% RSLogix 500 project XLT_EXP_BOTTOM.RSS, saved by version 11.00.00.00 %
PROJECT "LINCEBOT"    % processor: MicroLogix 1400 %

PROGRAM FILES
  LAD 2 "MAIN"  39 rungs  % Main Program Routine %
  LAD 6 "FEED"  16 rungs
  LAD 70 "OFFSETS"  29 rungs
  LAD 88 "TIMESWITCH"  2 rungs
  LAD 89 "SECONDS"  2 rungs
  LAD 90 "HSC"  9 rungs
  LAD 95 "HMI SET"  6 rungs
  LAD 100 "STI"  29 rungs
  LAD 102 "SPEED"  6 rungs
  LAD 104 "P ADJUST"  8 rungs
  LAD 110 "SHIFT"  7 rungs
  LAD 120 "SIM PARTS"  7 rungs
  LAD 121 "PARTDETECT"  4 rungs
  LAD 122 "OPTICWIDTH"  7 rungs
  LAD 123 "PART GAP"  10 rungs
  LAD 125 "OPTIC"  5 rungs
  LAD 130 "INS 1 TRIG"  24 rungs
  LAD 131 "INS 1 RSLT"  20 rungs
  LAD 150 "DEF HEAD"  10 rungs  % remove me %
  LAD 170 "XFER OUT"  6 rungs

DATA FILES
  O0 OUTPUT  11 elements
  I1 INPUT  11 elements
  S2 STATUS  66 elements
  B3 BINARY  14 elements
  T4 TIMER  40 elements
  C5 COUNTER  1 elements
  R6 CONTROL  10 elements
  N7 INTEGER  200 elements
  F8 FLOAT  100 elements
  B9 TOP BS DAT  256 elements
  B10 OLD_COM  1 elements
  B11 BOT BS DAT  256 elements
  L13  COUNTS  100 elements
  L23 NEW READ  100 elements
  L24 NEW WRITE  100 elements
  L42   52 elements
  B181 BLANK  128 elements  % used to wipe bs files %
  F182 TEST FLOAT  50 elements
  L183 TEST LONG  50 elements
  N184 TEST INTS  50 elements
  B185 TEST BITS  50 elements
  N186 HMI INTS  50 elements
  L187 HMI LONG  50 elements
  F188 HMI FLOAT  50 elements
  B189 HMI BITS  50 elements
  L190 COUNTS  50 elements
  B191 ERROR BITS  10 elements
  L192 SPD OFFSET  50 elements
  F193 SPD OFFSET  50 elements
  B194 GOOD BS  128 elements
  B195 NOERROR BS  128 elements
  B196 CTRL BITS  50 elements
  N197 CTRL INTS  50 elements
  B198 TRK BITS  50 elements
  L199 TRK LONG  50 elements
  N200 TRK INTS  50 elements
  L201 INS LONG  50 elements
  B202 INS BITS  50 elements
  N203 INS INTS  50 elements
  L204 CTRL LONG  50 elements
  F205 CTRL FLTS  50 elements

LADDER 2 "MAIN"    % Main Program Routine %
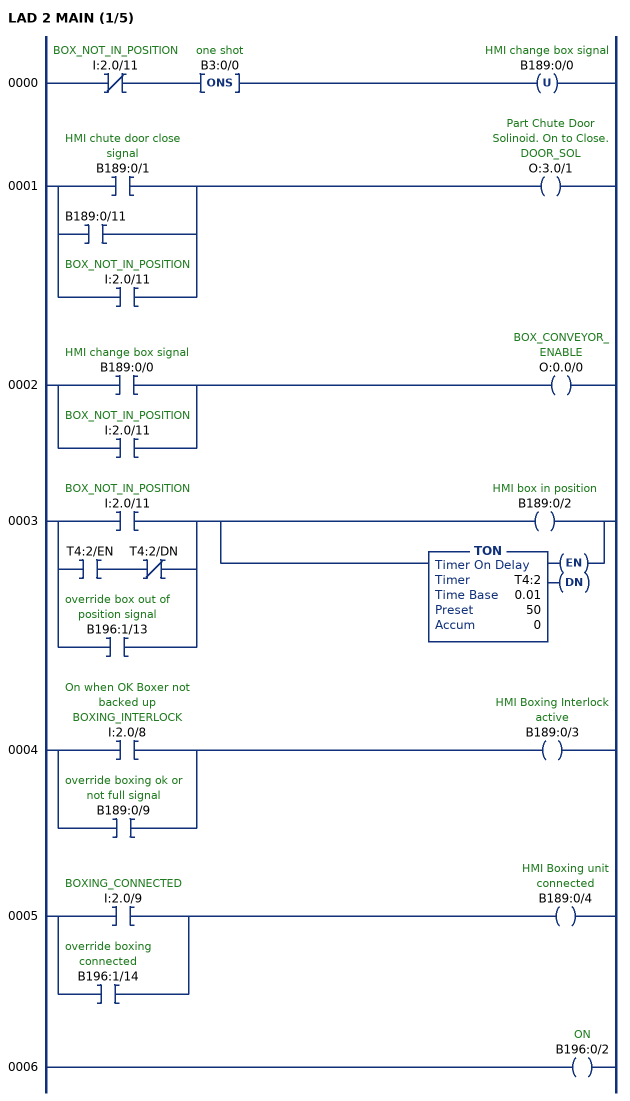
% Rung: 0 %
SOR XIO I:2.0/11 ONS B3:0/0 OTU B189:0/0 EOR
%   I:2.0/11  BOX_NOT_IN_POSITION %
%   B3:0/0  "one shot" %
%   B189:0/0  "HMI change box signal" %
% Rung: 1 %
SOR BST XIC B189:0/1 NXB XIC B189:0/11 NXB XIC I:2.0/11 BND OTE O:3.0/1 EOR
%   B189:0/1  "HMI chute door close signal" %
%   I:2.0/11  BOX_NOT_IN_POSITION %
%   O:3.0/1  DOOR_SOL  "Part Chute Door Solinoid. On to Close." %
% Rung: 2 %
SOR BST XIC B189:0/0 NXB XIC I:2.0/11 BND OTE O:0.0/0 EOR
%   B189:0/0  "HMI change box signal" %
%   I:2.0/11  BOX_NOT_IN_POSITION %
%   O:0.0/0  BOX_CONVEYOR_ENABLE %
% Rung: 3 %
SOR BST XIC I:2.0/11 NXB XIC T4:2/EN XIO T4:2/DN NXB XIC B196:1/13 BND BST OTE B189:0/2 NXB TON T4:2 0.01 50 0 BND EOR
%   I:2.0/11  BOX_NOT_IN_POSITION %
%   B196:1/13  "override box out of position signal" %
%   B189:0/2  "HMI box in position" %
% Rung: 4 %
SOR BST XIC I:2.0/8 NXB XIC B189:0/9 BND OTE B189:0/3 EOR
%   I:2.0/8  BOXING_INTERLOCK  "On when OK Boxer not backed up" %
%   B189:0/9  "override boxing ok or not full signal" %
%   B189:0/3  "HMI Boxing Interlock active" %
% Rung: 5 %
SOR BST XIC I:2.0/9 NXB XIC B196:1/14 BND OTE B189:0/4 EOR
%   I:2.0/9  BOXING_CONNECTED %
%   B196:1/14  "override boxing connected" %
%   B189:0/4  "HMI Boxing unit connected" %
% Rung: 6 %
SOR OTE B196:0/2 EOR
%   B196:0/2  ON %

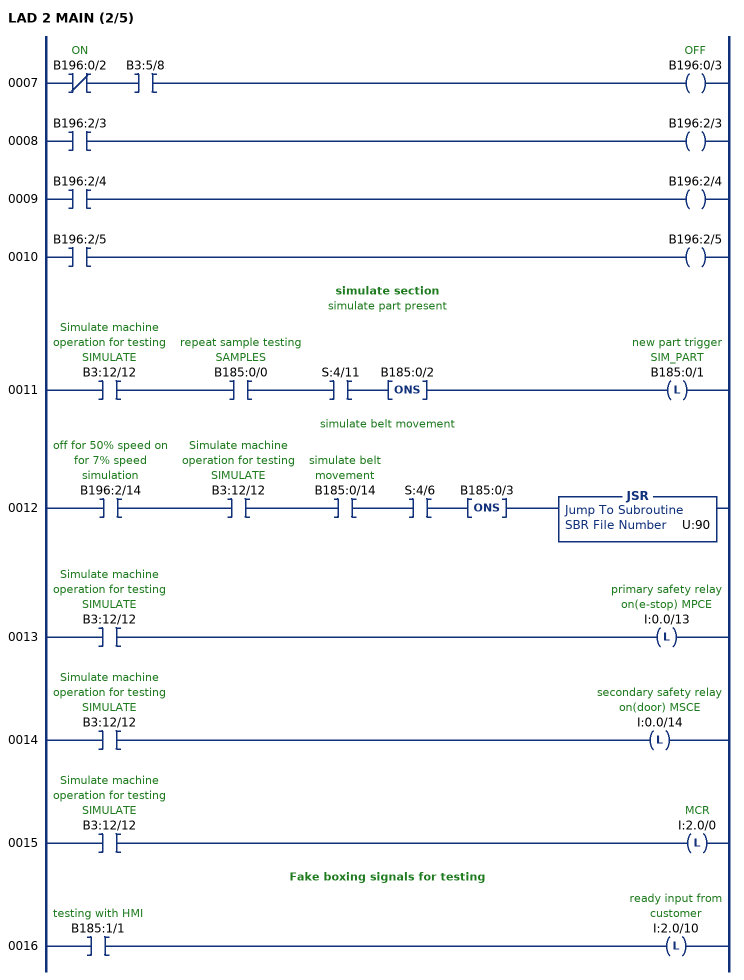
% Rung: 7 %
SOR XIO B196:0/2 XIC B3:5/8 OTE B196:0/3 EOR
%   B196:0/2  ON %
%   B196:0/3  OFF %
% Rung: 8 %
SOR XIC B196:2/3 OTE B196:2/3 EOR
% Rung: 9 %
SOR XIC B196:2/4 OTE B196:2/4 EOR
% Rung: 10 %
SOR XIC B196:2/5 OTE B196:2/5 EOR
% Rung: 11 %
% TITLE: simulate section %
% simulate part present %
SOR XIC B3:12/12 XIC B185:0/0 XIC S:4/11 ONS B185:0/2 OTL B185:0/1 EOR
%   B3:12/12  SIMULATE  "Simulate machine operation for testing" %
%   B185:0/0  SAMPLES  "repeat sample testing" %
%   B185:0/1  SIM_PART  "new part trigger" %
% Rung: 12 %
% simulate belt movement %
SOR XIC B196:2/14 XIC B3:12/12 XIC B185:0/14 XIC S:4/6 ONS B185:0/3 JSR U:90 EOR
%   B196:2/14  "off for 50% speed on for 7% speed simulation" %
%   B3:12/12  SIMULATE  "Simulate machine operation for testing" %
%   B185:0/14  "simulate belt movement" %
% Rung: 13 %
SOR XIC B3:12/12 OTL I:0.0/13 EOR
%   B3:12/12  SIMULATE  "Simulate machine operation for testing" %
%   I:0.0/13  MPCE  "primary safety relay on(e-stop)" %
% Rung: 14 %
SOR XIC B3:12/12 OTL I:0.0/14 EOR
%   B3:12/12  SIMULATE  "Simulate machine operation for testing" %
%   I:0.0/14  MSCE  "secondary safety relay on(door)" %
% Rung: 15 %
SOR XIC B3:12/12 OTL I:2.0/0 EOR
%   B3:12/12  SIMULATE  "Simulate machine operation for testing" %
%   I:2.0/0  MCR %
% Rung: 16 %
% TITLE: Fake boxing signals for testing %
SOR XIC B185:1/1 OTL I:2.0/10 EOR
%   B185:1/1  "testing with HMI" %
%   I:2.0/10  "ready input from customer" %

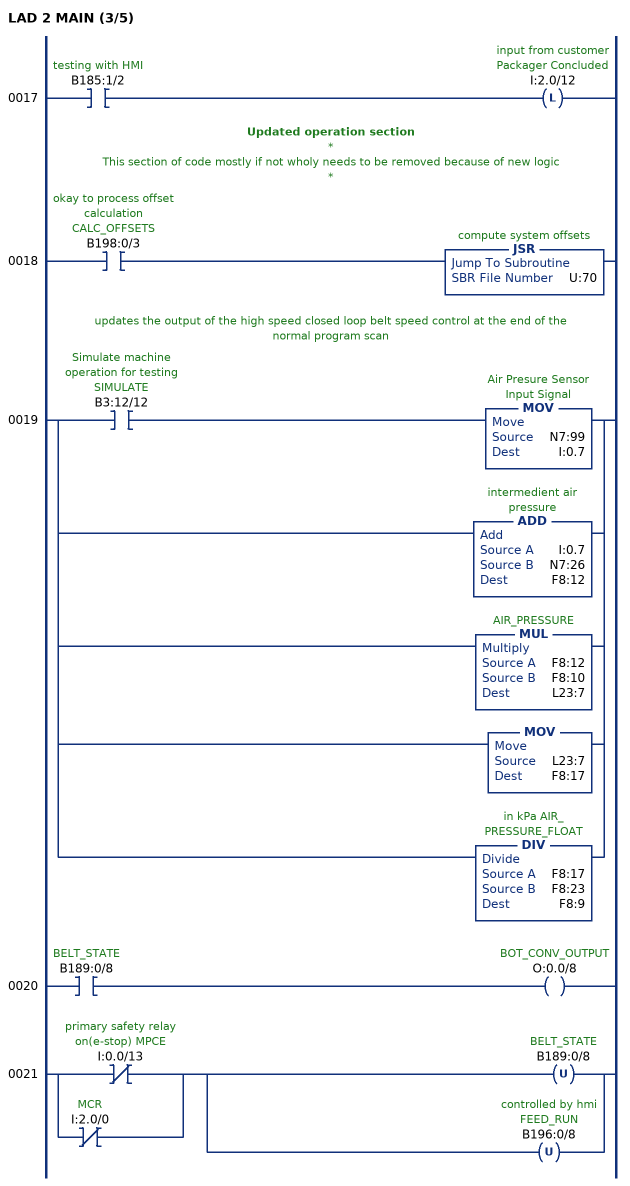
% Rung: 17 %
SOR XIC B185:1/2 OTL I:2.0/12 EOR
%   B185:1/2  "testing with HMI" %
%   I:2.0/12  "input from customer Packager Concluded" %
% Rung: 18 %
% TITLE: Updated operation section %
% *
% This section of code mostly if not wholy needs to be removed because of new logic
% * %
SOR XIC B198:0/3 JSR U:70 EOR
%   B198:0/3  CALC_OFFSETS  "okay to process offset calculation" %
%   U:70  "compute system offsets" %
% Rung: 19 %
% updates the output of the high speed closed loop belt speed control at the end of the normal program scan %
SOR BST XIC B3:12/12 MOV N7:99 I:0.7 NXB ADD I:0.7 N7:26 F8:12 NXB MUL F8:12 F8:10 L23:7 NXB MOV L23:7 F8:17 NXB DIV F8:17 F8:23 F8:9 BND EOR
%   B3:12/12  SIMULATE  "Simulate machine operation for testing" %
%   I:0.7  "Air Presure Sensor Input Signal" %
%   N7:26  MAIN_AIR_OFFSET  "Main Air Offset old machine -398 new machine 0" %
%   F8:12  "intermedient air pressure" %
%   F8:10  AIR_MULTIPLIER_BAR  "Air Multiplier (BAR)" %
%   L23:7  AIR_PRESSURE %
%   F8:9  AIR_PRESSURE_FLOAT  "in kPa" %
% Rung: 20 %
SOR XIC B189:0/8 OTE O:0.0/8 EOR
%   B189:0/8  BELT_STATE %
%   O:0.0/8  BOT_CONV_OUTPUT %
% Rung: 21 %
SOR BST XIO I:0.0/13 NXB XIO I:2.0/0 BND BST OTU B189:0/8 NXB OTU B196:0/8 BND EOR
%   I:0.0/13  MPCE  "primary safety relay on(e-stop)" %
%   I:2.0/0  MCR %
%   B189:0/8  BELT_STATE %
%   B196:0/8  FEED_RUN  "controlled by hmi" %

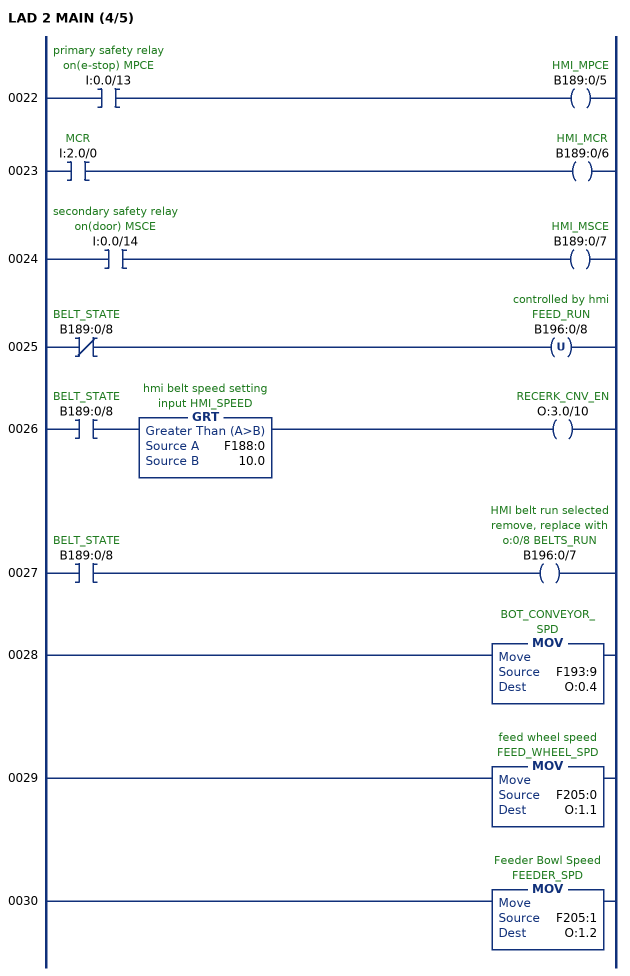
% Rung: 22 %
SOR XIC I:0.0/13 OTE B189:0/5 EOR
%   I:0.0/13  MPCE  "primary safety relay on(e-stop)" %
%   B189:0/5  HMI_MPCE %
% Rung: 23 %
SOR XIC I:2.0/0 OTE B189:0/6 EOR
%   I:2.0/0  MCR %
%   B189:0/6  HMI_MCR %
% Rung: 24 %
SOR XIC I:0.0/14 OTE B189:0/7 EOR
%   I:0.0/14  MSCE  "secondary safety relay on(door)" %
%   B189:0/7  HMI_MSCE %
% Rung: 25 %
SOR XIO B189:0/8 OTU B196:0/8 EOR
%   B189:0/8  BELT_STATE %
%   B196:0/8  FEED_RUN  "controlled by hmi" %
% Rung: 26 %
SOR XIC B189:0/8 GRT F188:0 10.0 OTE O:3.0/10 EOR
%   B189:0/8  BELT_STATE %
%   F188:0  HMI_SPEED  "hmi belt speed setting input" %
%   O:3.0/10  RECERK_CNV_EN %
% Rung: 27 %
SOR XIC B189:0/8 OTE B196:0/7 EOR
%   B189:0/8  BELT_STATE %
%   B196:0/7  BELTS_RUN  "HMI belt run selected remove, replace with o:0/8" %
% Rung: 28 %
SOR MOV F193:9 O:0.4 EOR
%   F193:9  CTRLED_SCALED_VALUE %
%   O:0.4  BOT_CONVEYOR_SPD %
% Rung: 29 %
SOR MOV F205:0 O:1.1 EOR
%   F205:0  "feed wheel" %
%   O:1.1  FEED_WHEEL_SPD  "feed wheel speed" %
% Rung: 30 %
SOR MOV F205:1 O:1.2 EOR
%   F205:1  "feed bowl" %
%   O:1.2  FEEDER_SPD  "Feeder Bowl Speed" %

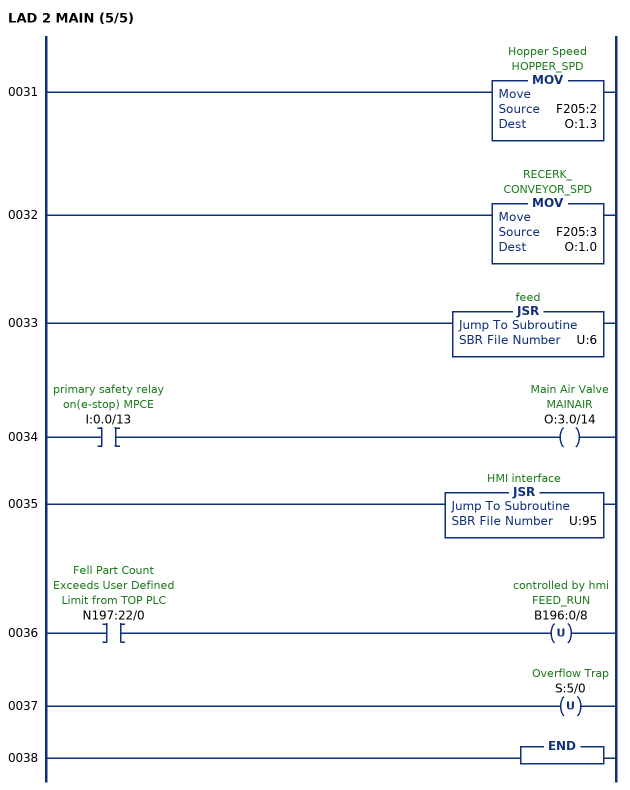
% Rung: 31 %
SOR MOV F205:2 O:1.3 EOR
%   F205:2  "hopper" %
%   O:1.3  HOPPER_SPD  "Hopper Speed" %
% Rung: 32 %
SOR MOV F205:3 O:1.0 EOR
%   F205:3  "recerk" %
%   O:1.0  RECERK_CONVEYOR_SPD %
% Rung: 33 %
SOR JSR U:6 EOR
%   U:6  "feed" %
% Rung: 34 %
SOR XIC I:0.0/13 OTE O:3.0/14 EOR
%   I:0.0/13  MPCE  "primary safety relay on(e-stop)" %
%   O:3.0/14  MAINAIR  "Main Air Valve" %
% Rung: 35 %
SOR JSR U:95 EOR
%   U:95  "HMI interface" %
% Rung: 36 %
SOR XIC N197:22/0 OTU B196:0/8 EOR
%   N197:22/0  "Fell Part Count Exceeds User Defined Limit from TOP PLC" %
%   B196:0/8  FEED_RUN  "controlled by hmi" %
% Rung: 37 %
SOR OTU S:5/0 EOR
%   S:5/0  "Overflow Trap" %
% Rung: 38 %
SOR END EOR

LADDER 6 "FEED"
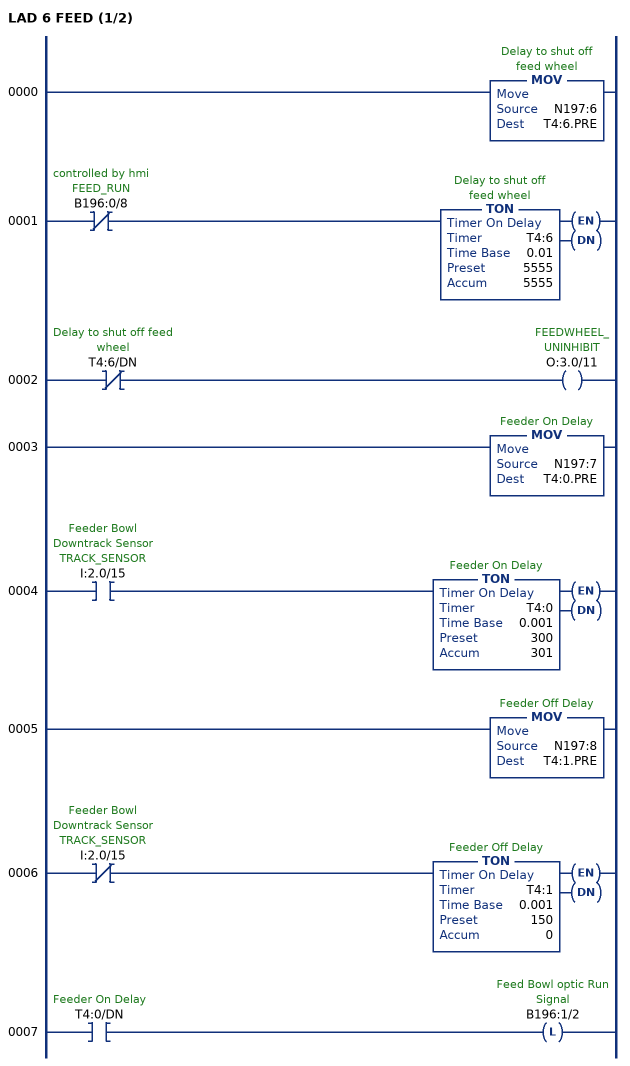
% Rung: 0 %
SOR MOV N197:6 T4:6.PRE EOR
%   N197:6  "feed wheel time delayed shutoff" %
%   T4:6  "Delay to shut off feed wheel" %
% Rung: 1 %
SOR XIO B196:0/8 TON T4:6 0.01 5555 5555 EOR
%   B196:0/8  FEED_RUN  "controlled by hmi" %
%   T4:6  "Delay to shut off feed wheel" %
% Rung: 2 %
SOR XIO T4:6/DN OTE O:3.0/11 EOR
%   T4:6  "Delay to shut off feed wheel" %
%   O:3.0/11  FEEDWHEEL_UNINHIBIT %
% Rung: 3 %
SOR MOV N197:7 T4:0.PRE EOR
%   N197:7  "down track on delay" %
%   T4:0  "Feeder On Delay" %
% Rung: 4 %
SOR XIC I:2.0/15 TON T4:0 0.001 300 301 EOR
%   I:2.0/15  TRACK_SENSOR  "Feeder Bowl Downtrack Sensor" %
%   T4:0  "Feeder On Delay" %
% Rung: 5 %
SOR MOV N197:8 T4:1.PRE EOR
%   N197:8  "down track off delay" %
%   T4:1  "Feeder Off Delay" %
% Rung: 6 %
SOR XIO I:2.0/15 TON T4:1 0.001 150 0 EOR
%   I:2.0/15  TRACK_SENSOR  "Feeder Bowl Downtrack Sensor" %
%   T4:1  "Feeder Off Delay" %
% Rung: 7 %
SOR XIC T4:0/DN OTL B196:1/2 EOR
%   T4:0  "Feeder On Delay" %
%   B196:1/2  "Feed Bowl optic Run Signal" %

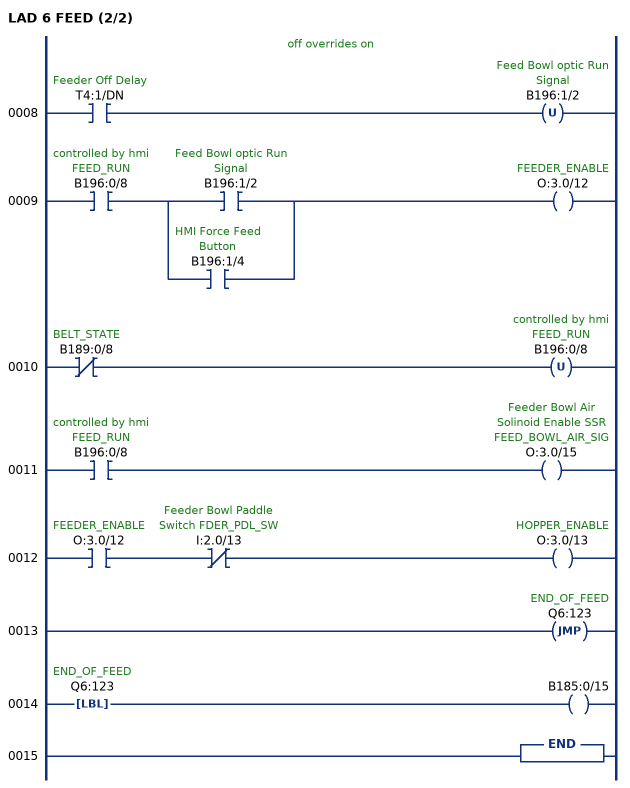
% Rung: 8 %
% off overrides on %
SOR XIC T4:1/DN OTU B196:1/2 EOR
%   T4:1  "Feeder Off Delay" %
%   B196:1/2  "Feed Bowl optic Run Signal" %
% Rung: 9 %
SOR XIC B196:0/8 BST XIC B196:1/2 NXB XIC B196:1/4 BND OTE O:3.0/12 EOR
%   B196:0/8  FEED_RUN  "controlled by hmi" %
%   B196:1/2  "Feed Bowl optic Run Signal" %
%   B196:1/4  "HMI Force Feed Button" %
%   O:3.0/12  FEEDER_ENABLE %
% Rung: 10 %
SOR XIO B189:0/8 OTU B196:0/8 EOR
%   B189:0/8  BELT_STATE %
%   B196:0/8  FEED_RUN  "controlled by hmi" %
% Rung: 11 %
SOR XIC B196:0/8 OTE O:3.0/15 EOR
%   B196:0/8  FEED_RUN  "controlled by hmi" %
%   O:3.0/15  FEED_BOWL_AIR_SIG  "Feeder Bowl Air Solinoid Enable SSR" %
% Rung: 12 %
SOR XIC O:3.0/12 XIO I:2.0/13 OTE O:3.0/13 EOR
%   O:3.0/12  FEEDER_ENABLE %
%   I:2.0/13  FDER_PDL_SW  "Feeder Bowl Paddle Switch" %
%   O:3.0/13  HOPPER_ENABLE %
% Rung: 13 %
SOR JMP Q6:123 EOR
%   Q6:123  END_OF_FEED %
% Rung: 14 %
SOR LBL Q6:123 OTE B185:0/15 EOR
%   Q6:123  END_OF_FEED %
% Rung: 15 %
SOR END EOR

LADDER 70 "OFFSETS"
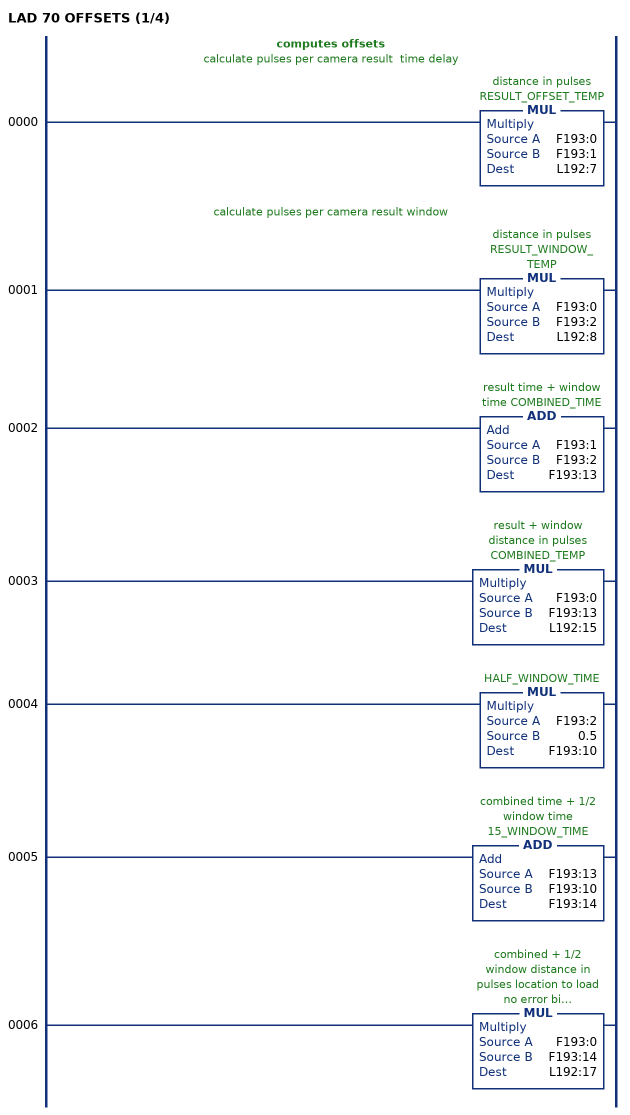
% Rung: 0 %
% TITLE: computes offsets %
% calculate pulses per camera result  time delay %
SOR MUL F193:0 F193:1 L192:7 EOR
%   F193:0  SPD  "speed calculation result (PPS)" %
%   F193:1  RESULT_TIME_F  "Seconds" %
%   L192:7  RESULT_OFFSET_TEMP  "distance in pulses" %
% Rung: 1 %
% calculate pulses per camera result window %
SOR MUL F193:0 F193:2 L192:8 EOR
%   F193:0  SPD  "speed calculation result (PPS)" %
%   F193:2  WINDOW_TIME_F  "seconds" %
%   L192:8  RESULT_WINDOW_TEMP  "distance in pulses" %
% Rung: 2 %
SOR ADD F193:1 F193:2 F193:13 EOR
%   F193:1  RESULT_TIME_F  "Seconds" %
%   F193:2  WINDOW_TIME_F  "seconds" %
%   F193:13  COMBINED_TIME  "result time + window time" %
% Rung: 3 %
SOR MUL F193:0 F193:13 L192:15 EOR
%   F193:0  SPD  "speed calculation result (PPS)" %
%   F193:13  COMBINED_TIME  "result time + window time" %
%   L192:15  COMBINED_TEMP  "result + window distance in pulses" %
% Rung: 4 %
SOR MUL F193:2 0.5 F193:10 EOR
%   F193:2  WINDOW_TIME_F  "seconds" %
%   F193:10  HALF_WINDOW_TIME %
% Rung: 5 %
SOR ADD F193:13 F193:10 F193:14 EOR
%   F193:13  COMBINED_TIME  "result time + window time" %
%   F193:10  HALF_WINDOW_TIME %
%   F193:14  15_WINDOW_TIME  "combined time + 1/2 window time" %
% Rung: 6 %
SOR MUL F193:0 F193:14 L192:17 EOR
%   F193:0  SPD  "speed calculation result (PPS)" %
%   F193:14  15_WINDOW_TIME  "combined time + 1/2 window time" %
%   L192:17  15_WINDOW_TEMP  "combined + 1/2 window distance in pulses location to load no error bit" %

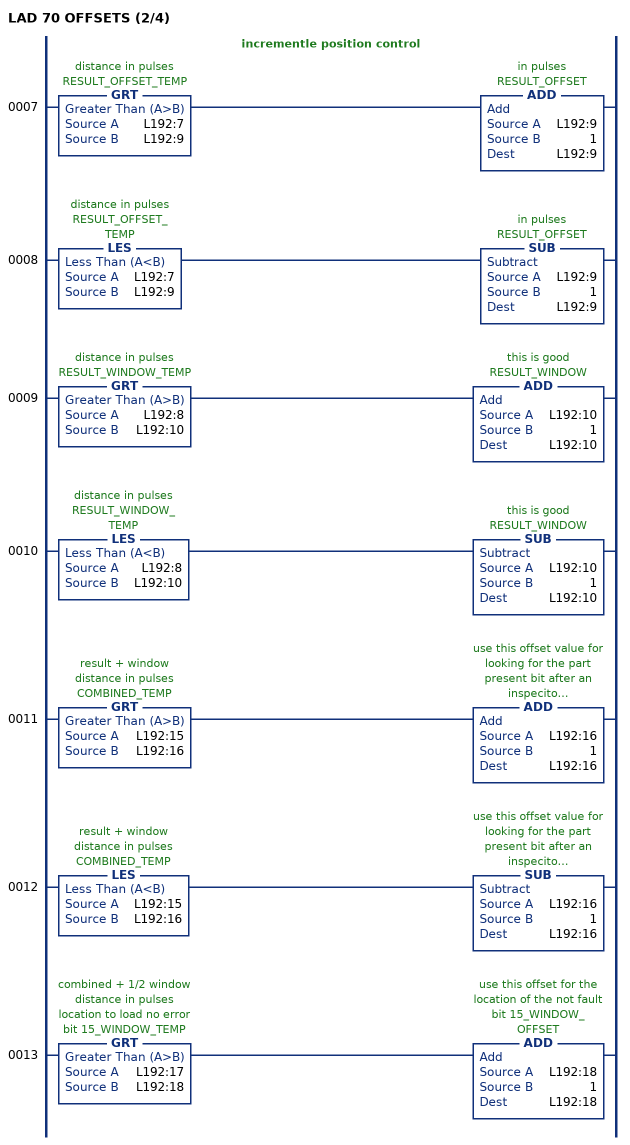
% Rung: 7 %
% TITLE: incrementle position control %
SOR GRT L192:7 L192:9 ADD L192:9 1 L192:9 EOR
%   L192:7  RESULT_OFFSET_TEMP  "distance in pulses" %
%   L192:9  RESULT_OFFSET  "in pulses" %
% Rung: 8 %
SOR LES L192:7 L192:9 SUB L192:9 1 L192:9 EOR
%   L192:7  RESULT_OFFSET_TEMP  "distance in pulses" %
%   L192:9  RESULT_OFFSET  "in pulses" %
% Rung: 9 %
SOR GRT L192:8 L192:10 ADD L192:10 1 L192:10 EOR
%   L192:8  RESULT_WINDOW_TEMP  "distance in pulses" %
%   L192:10  RESULT_WINDOW  "this is good" %
% Rung: 10 %
SOR LES L192:8 L192:10 SUB L192:10 1 L192:10 EOR
%   L192:8  RESULT_WINDOW_TEMP  "distance in pulses" %
%   L192:10  RESULT_WINDOW  "this is good" %
% Rung: 11 %
SOR GRT L192:15 L192:16 ADD L192:16 1 L192:16 EOR
%   L192:15  COMBINED_TEMP  "result + window distance in pulses" %
%   L192:16  COMBINED_OFFSET  "use this offset value for looking for the part present bit after an inspeciton" %
% Rung: 12 %
SOR LES L192:15 L192:16 SUB L192:16 1 L192:16 EOR
%   L192:15  COMBINED_TEMP  "result + window distance in pulses" %
%   L192:16  COMBINED_OFFSET  "use this offset value for looking for the part present bit after an inspeciton" %
% Rung: 13 %
SOR GRT L192:17 L192:18 ADD L192:18 1 L192:18 EOR
%   L192:17  15_WINDOW_TEMP  "combined + 1/2 window distance in pulses location to load no error bit" %
%   L192:18  15_WINDOW_OFFSET  "use this offset for the location of the not fault bit" %

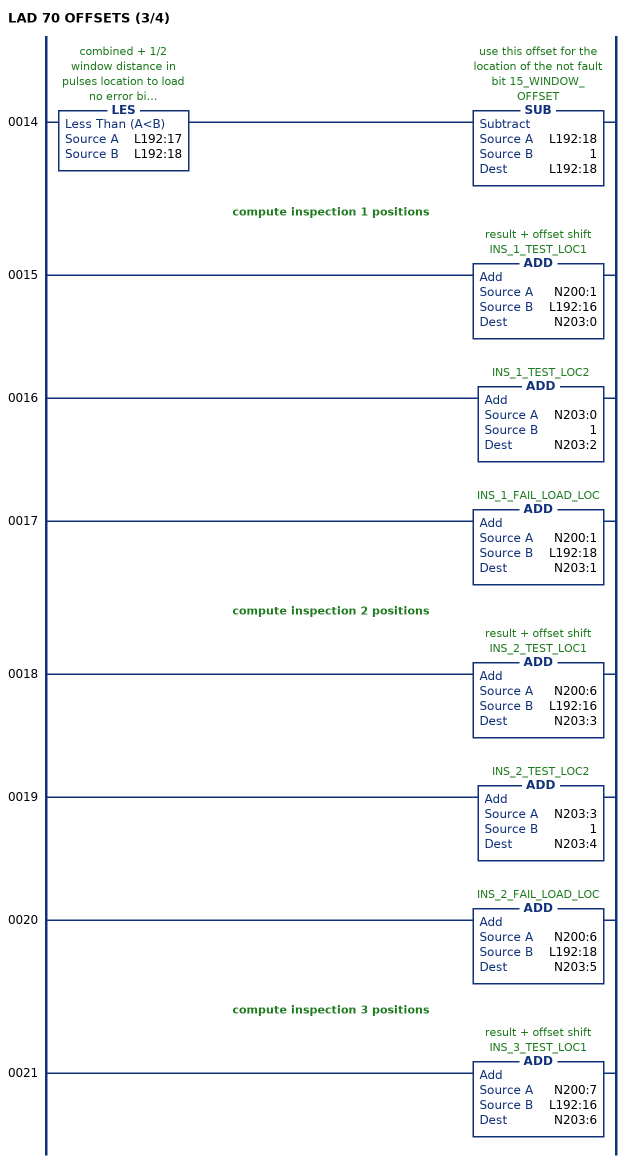
% Rung: 14 %
SOR LES L192:17 L192:18 SUB L192:18 1 L192:18 EOR
%   L192:17  15_WINDOW_TEMP  "combined + 1/2 window distance in pulses location to load no error bit" %
%   L192:18  15_WINDOW_OFFSET  "use this offset for the location of the not fault bit" %
% Rung: 15 %
% TITLE: compute inspection 1 positions %
SOR ADD N200:1 L192:16 N203:0 EOR
%   N200:1  INS_1_TRIG_LOC %
%   L192:16  COMBINED_OFFSET  "use this offset value for looking for the part present bit after an inspeciton" %
%   N203:0  INS_1_TEST_LOC1  "result + offset shift" %
% Rung: 16 %
SOR ADD N203:0 1 N203:2 EOR
%   N203:0  INS_1_TEST_LOC1  "result + offset shift" %
%   N203:2  INS_1_TEST_LOC2 %
% Rung: 17 %
SOR ADD N200:1 L192:18 N203:1 EOR
%   N200:1  INS_1_TRIG_LOC %
%   L192:18  15_WINDOW_OFFSET  "use this offset for the location of the not fault bit" %
%   N203:1  INS_1_FAIL_LOAD_LOC %
% Rung: 18 %
% TITLE: compute inspection 2 positions %
SOR ADD N200:6 L192:16 N203:3 EOR
%   N200:6  INS_2_TRIG_LOC %
%   L192:16  COMBINED_OFFSET  "use this offset value for looking for the part present bit after an inspeciton" %
%   N203:3  INS_2_TEST_LOC1  "result + offset shift" %
% Rung: 19 %
SOR ADD N203:3 1 N203:4 EOR
%   N203:3  INS_2_TEST_LOC1  "result + offset shift" %
%   N203:4  INS_2_TEST_LOC2 %
% Rung: 20 %
SOR ADD N200:6 L192:18 N203:5 EOR
%   N200:6  INS_2_TRIG_LOC %
%   L192:18  15_WINDOW_OFFSET  "use this offset for the location of the not fault bit" %
%   N203:5  INS_2_FAIL_LOAD_LOC %
% Rung: 21 %
% TITLE: compute inspection 3 positions %
SOR ADD N200:7 L192:16 N203:6 EOR
%   N200:7  INS_3_TRIG_LOC %
%   L192:16  COMBINED_OFFSET  "use this offset value for looking for the part present bit after an inspeciton" %
%   N203:6  INS_3_TEST_LOC1  "result + offset shift" %

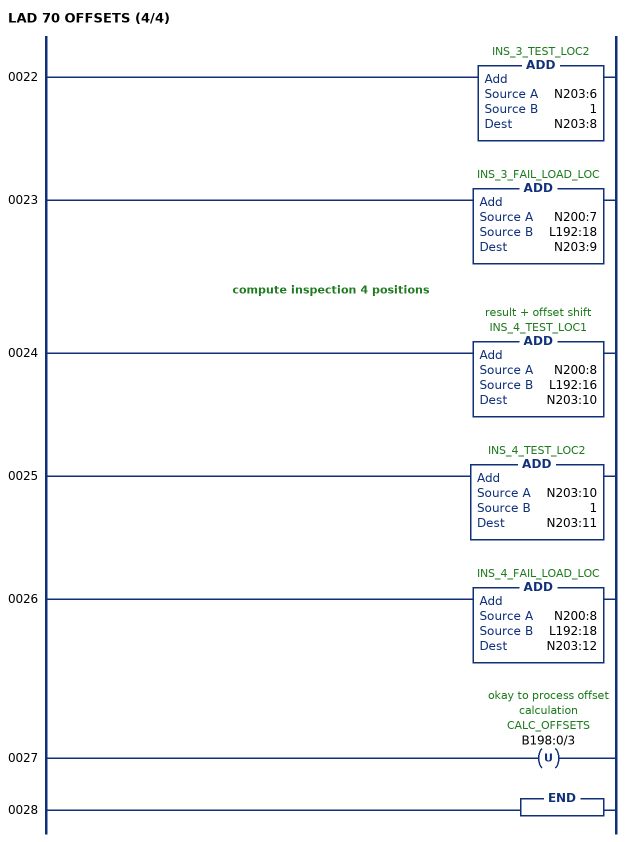
% Rung: 22 %
SOR ADD N203:6 1 N203:8 EOR
%   N203:6  INS_3_TEST_LOC1  "result + offset shift" %
%   N203:8  INS_3_TEST_LOC2 %
% Rung: 23 %
SOR ADD N200:7 L192:18 N203:9 EOR
%   N200:7  INS_3_TRIG_LOC %
%   L192:18  15_WINDOW_OFFSET  "use this offset for the location of the not fault bit" %
%   N203:9  INS_3_FAIL_LOAD_LOC %
% Rung: 24 %
% TITLE: compute inspection 4 positions %
SOR ADD N200:8 L192:16 N203:10 EOR
%   N200:8  INS_4_TRIG_LOC %
%   L192:16  COMBINED_OFFSET  "use this offset value for looking for the part present bit after an inspeciton" %
%   N203:10  INS_4_TEST_LOC1  "result + offset shift" %
% Rung: 25 %
SOR ADD N203:10 1 N203:11 EOR
%   N203:10  INS_4_TEST_LOC1  "result + offset shift" %
%   N203:11  INS_4_TEST_LOC2 %
% Rung: 26 %
SOR ADD N200:8 L192:18 N203:12 EOR
%   N200:8  INS_4_TRIG_LOC %
%   L192:18  15_WINDOW_OFFSET  "use this offset for the location of the not fault bit" %
%   N203:12  INS_4_FAIL_LOAD_LOC %
% Rung: 27 %
SOR OTU B198:0/3 EOR
%   B198:0/3  CALC_OFFSETS  "okay to process offset calculation" %
% Rung: 28 %
SOR END EOR

LADDER 88 "TIMESWITCH"
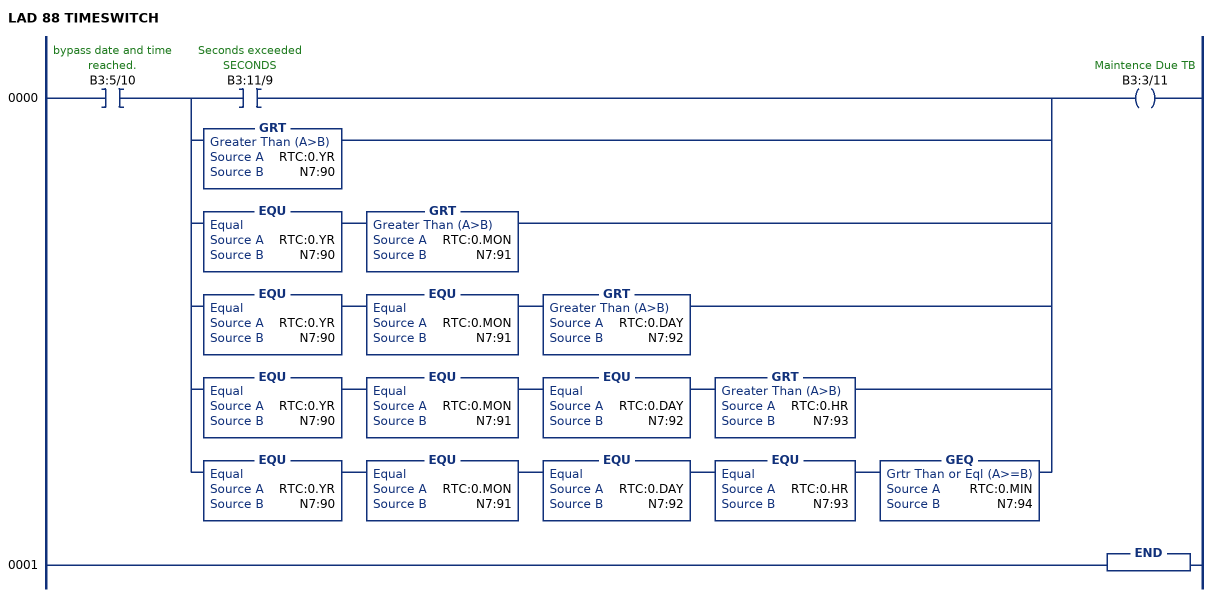
% Rung: 0 %
SOR XIC B3:5/10 BST XIC B3:11/9 NXB GRT RTC:0.YR N7:90 NXB EQU RTC:0.YR N7:90 GRT RTC:0.MON N7:91 NXB EQU RTC:0.YR N7:90 EQU RTC:0.MON N7:91 GRT RTC:0.DAY N7:92 NXB EQU RTC:0.YR N7:90 EQU RTC:0.MON N7:91 EQU RTC:0.DAY N7:92 GRT RTC:0.HR N7:93 NXB EQU RTC:0.YR N7:90 EQU RTC:0.MON N7:91 EQU RTC:0.DAY N7:92 EQU RTC:0.HR N7:93 GEQ RTC:0.MIN N7:94 BND OTE B3:3/11 EOR
%   B3:5/10  "bypass date and time reached." %
%   B3:11/9  SECONDS  "Seconds exceeded" %
%   N7:90  RTC %
%   B3:3/11  TB  "Maintence Due" %
% Rung: 1 %
SOR END EOR

LADDER 89 "SECONDS"
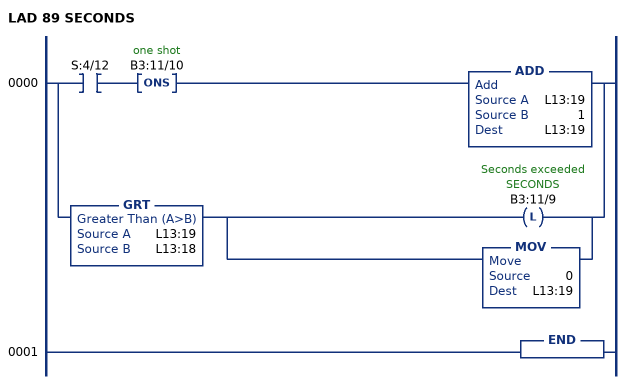
% Rung: 0 %
SOR BST XIC S:4/12 ONS B3:11/10 ADD L13:19 1 L13:19 NXB GRT L13:19 L13:18 BST OTL B3:11/9 NXB MOV 0 L13:19 BND BND EOR
%   B3:11/10  "one shot" %
%   L13:18  MAX %
%   B3:11/9  SECONDS  "Seconds exceeded" %
% Rung: 1 %
SOR END EOR

LADDER 90 "HSC"
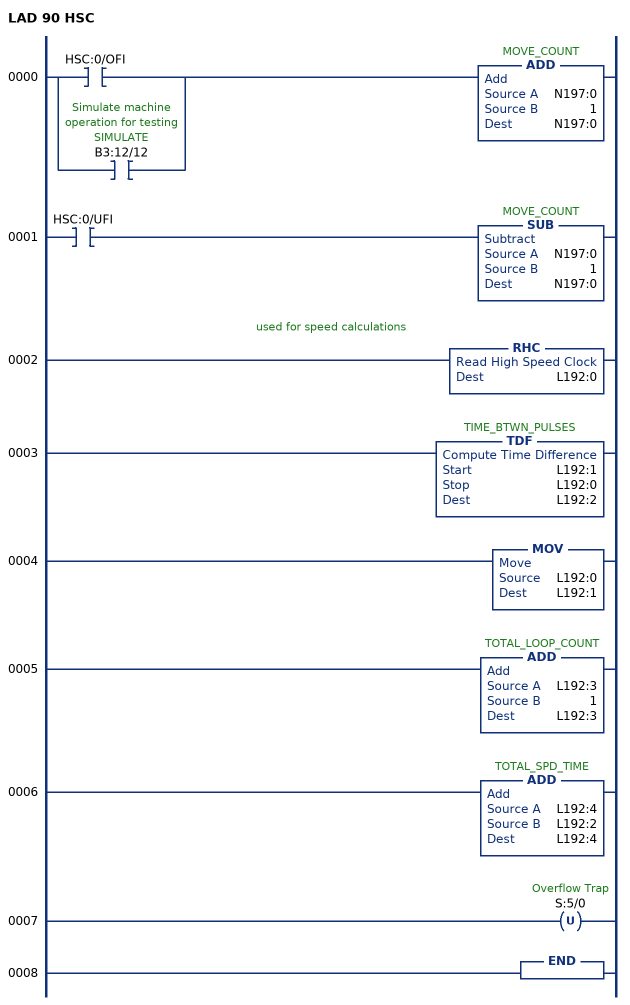
% Rung: 0 %
SOR BST XIC HSC:0/OFI NXB XIC B3:12/12 BND ADD N197:0 1 N197:0 EOR
%   B3:12/12  SIMULATE  "Simulate machine operation for testing" %
%   N197:0  MOVE_COUNT %
% Rung: 1 %
SOR XIC HSC:0/UFI SUB N197:0 1 N197:0 EOR
%   N197:0  MOVE_COUNT %
% Rung: 2 %
% used for speed calculations %
SOR RHC L192:0 EOR
% Rung: 3 %
SOR TDF L192:1 L192:0 L192:2 EOR
%   L192:2  TIME_BTWN_PULSES %
% Rung: 4 %
SOR MOV L192:0 L192:1 EOR
% Rung: 5 %
SOR ADD L192:3 1 L192:3 EOR
%   L192:3  TOTAL_LOOP_COUNT %
% Rung: 6 %
SOR ADD L192:4 L192:2 L192:4 EOR
%   L192:4  TOTAL_SPD_TIME %
%   L192:2  TIME_BTWN_PULSES %
% Rung: 7 %
SOR OTU S:5/0 EOR
%   S:5/0  "Overflow Trap" %
% Rung: 8 %
SOR END EOR

LADDER 95 "HMI SET"
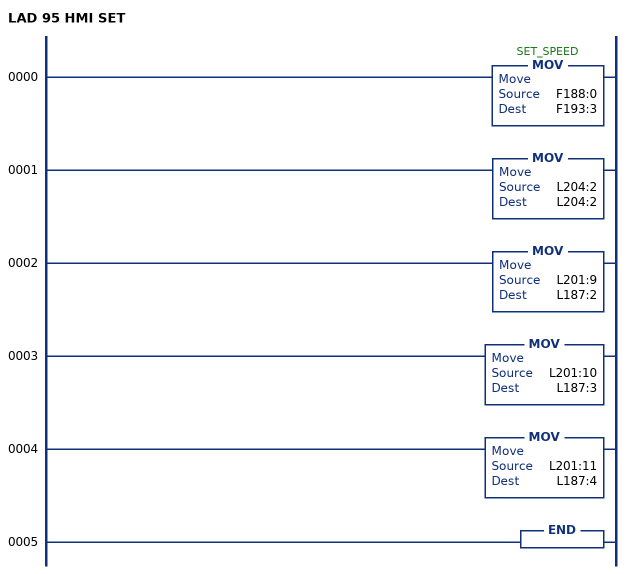
% Rung: 0 %
SOR MOV F188:0 F193:3 EOR
%   F188:0  HMI_SPEED  "hmi belt speed setting input" %
%   F193:3  SET_SPEED %
% Rung: 1 %
SOR MOV L204:2 L204:2 EOR
% Rung: 2 %
SOR MOV L201:9 L187:2 EOR
% Rung: 3 %
SOR MOV L201:10 L187:3 EOR
%   L201:10  "movement from virtual (pos, add)" %
% Rung: 4 %
SOR MOV L201:11 L187:4 EOR
% Rung: 5 %
SOR END EOR

LADDER 100 "STI"
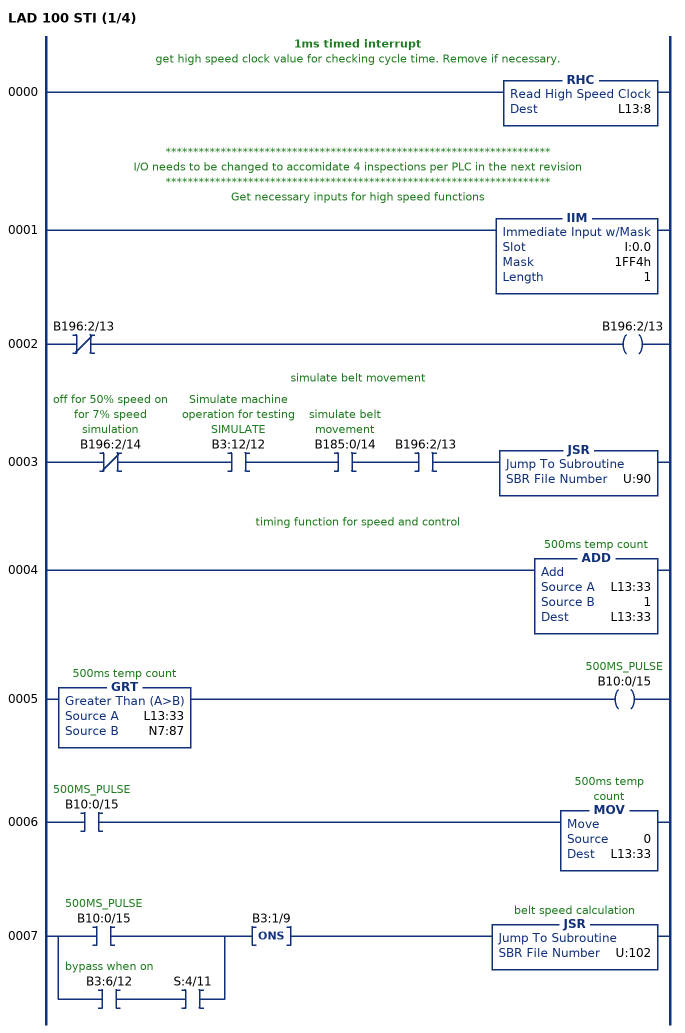
% Rung: 0 %
% TITLE: 1ms timed interrupt %
% get high speed clock value for checking cycle time. Remove if necessary. %
SOR RHC L13:8 EOR
% Rung: 1 %
% **********************************************************************
% 
% I/O needs to be changed to accomidate 4 inspections per PLC in the next revision
% 
% **********************************************************************
% 
% Get necessary inputs for high speed functions %
SOR IIM I:0.0 1FF4h 1 EOR
% Rung: 2 %
SOR XIO B196:2/13 OTE B196:2/13 EOR
% Rung: 3 %
% simulate belt movement %
SOR XIO B196:2/14 XIC B3:12/12 XIC B185:0/14 XIC B196:2/13 JSR U:90 EOR
%   B196:2/14  "off for 50% speed on for 7% speed simulation" %
%   B3:12/12  SIMULATE  "Simulate machine operation for testing" %
%   B185:0/14  "simulate belt movement" %
% Rung: 4 %
% timing function for speed and control %
SOR ADD L13:33 1 L13:33 EOR
%   L13:33  "500ms temp count" %
% Rung: 5 %
SOR GRT L13:33 N7:87 OTE B10:0/15 EOR
%   L13:33  "500ms temp count" %
%   B10:0/15  500MS_PULSE %
% Rung: 6 %
SOR XIC B10:0/15 MOV 0 L13:33 EOR
%   B10:0/15  500MS_PULSE %
%   L13:33  "500ms temp count" %
% Rung: 7 %
SOR BST XIC B10:0/15 NXB XIC B3:6/12 XIC S:4/11 BND ONS B3:1/9 JSR U:102 EOR
%   B10:0/15  500MS_PULSE %
%   B3:6/12  "bypass when on" %
%   U:102  "belt speed calculation" %

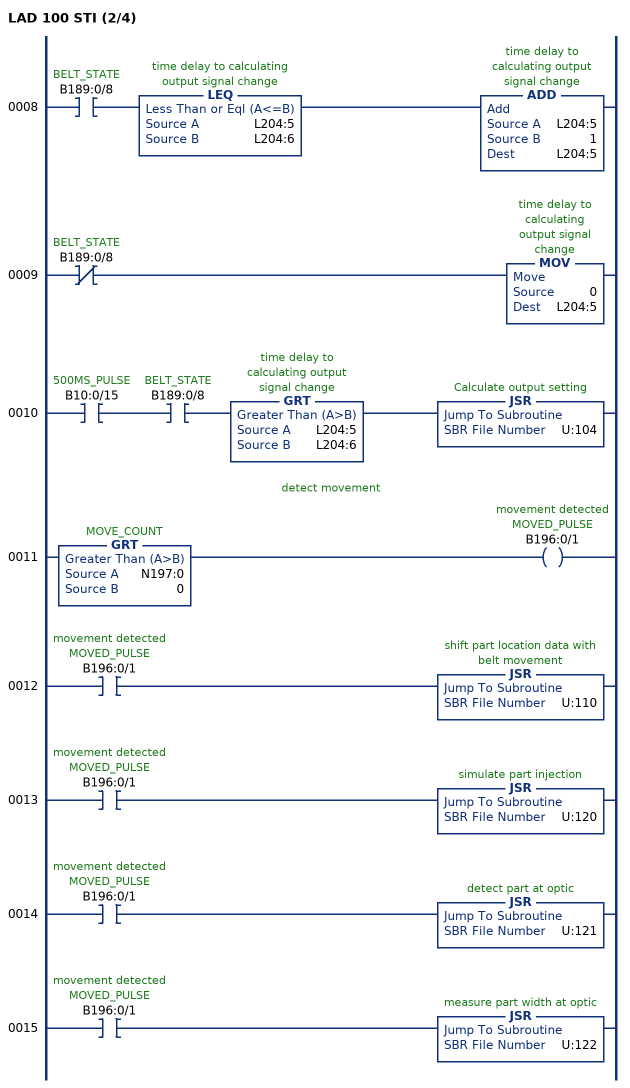
% Rung: 8 %
SOR XIC B189:0/8 LEQ L204:5 L204:6 ADD L204:5 1 L204:5 EOR
%   B189:0/8  BELT_STATE %
%   L204:5  "time delay to calculating output signal change" %
%   L204:6  "belt start delay time" %
% Rung: 9 %
SOR XIO B189:0/8 MOV 0 L204:5 EOR
%   B189:0/8  BELT_STATE %
%   L204:5  "time delay to calculating output signal change" %
% Rung: 10 %
SOR XIC B10:0/15 XIC B189:0/8 GRT L204:5 L204:6 JSR U:104 EOR
%   B10:0/15  500MS_PULSE %
%   B189:0/8  BELT_STATE %
%   L204:5  "time delay to calculating output signal change" %
%   L204:6  "belt start delay time" %
%   U:104  "Calculate output setting" %
% Rung: 11 %
% detect movement %
SOR GRT N197:0 0 OTE B196:0/1 EOR
%   N197:0  MOVE_COUNT %
%   B196:0/1  MOVED_PULSE  "movement detected" %
% Rung: 12 %
SOR XIC B196:0/1 JSR U:110 EOR
%   B196:0/1  MOVED_PULSE  "movement detected" %
%   U:110  "shift part location data with belt movement" %
% Rung: 13 %
SOR XIC B196:0/1 JSR U:120 EOR
%   B196:0/1  MOVED_PULSE  "movement detected" %
%   U:120  "simulate part injection" %
% Rung: 14 %
SOR XIC B196:0/1 JSR U:121 EOR
%   B196:0/1  MOVED_PULSE  "movement detected" %
%   U:121  "detect part at optic" %
% Rung: 15 %
SOR XIC B196:0/1 JSR U:122 EOR
%   B196:0/1  MOVED_PULSE  "movement detected" %
%   U:122  "measure part width at optic" %

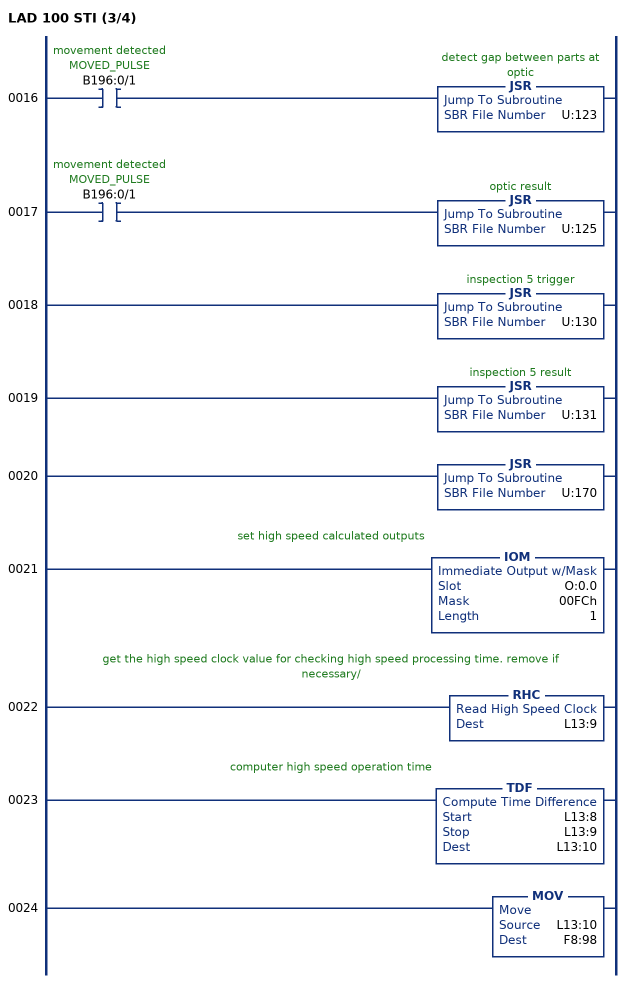
% Rung: 16 %
SOR XIC B196:0/1 JSR U:123 EOR
%   B196:0/1  MOVED_PULSE  "movement detected" %
%   U:123  "detect gap between parts at optic" %
% Rung: 17 %
SOR XIC B196:0/1 JSR U:125 EOR
%   B196:0/1  MOVED_PULSE  "movement detected" %
%   U:125  "optic result" %
% Rung: 18 %
SOR JSR U:130 EOR
%   U:130  "inspection 5 trigger" %
% Rung: 19 %
SOR JSR U:131 EOR
%   U:131  "inspection 5 result" %
% Rung: 20 %
SOR JSR U:170 EOR
% Rung: 21 %
% set high speed calculated outputs %
SOR IOM O:0.0 00FCh 1 EOR
% Rung: 22 %
% get the high speed clock value for checking high speed processing time. remove if necessary/ %
SOR RHC L13:9 EOR
% Rung: 23 %
% computer high speed operation time %
SOR TDF L13:8 L13:9 L13:10 EOR
% Rung: 24 %
SOR MOV L13:10 F8:98 EOR

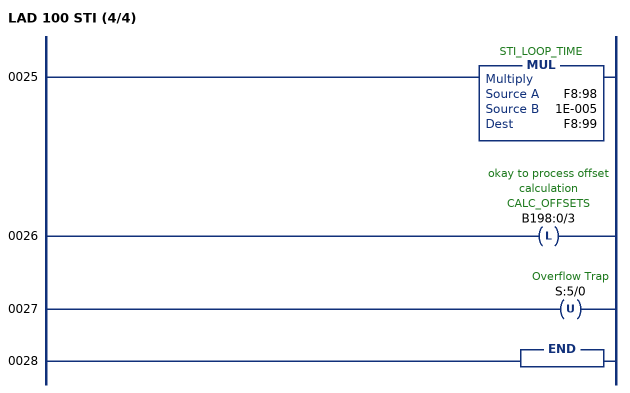
% Rung: 25 %
SOR MUL F8:98 1E-005 F8:99 EOR
%   F8:99  STI_LOOP_TIME %
% Rung: 26 %
SOR OTL B198:0/3 EOR
%   B198:0/3  CALC_OFFSETS  "okay to process offset calculation" %
% Rung: 27 %
SOR OTU S:5/0 EOR
%   S:5/0  "Overflow Trap" %
% Rung: 28 %
SOR END EOR

LADDER 102 "SPEED"
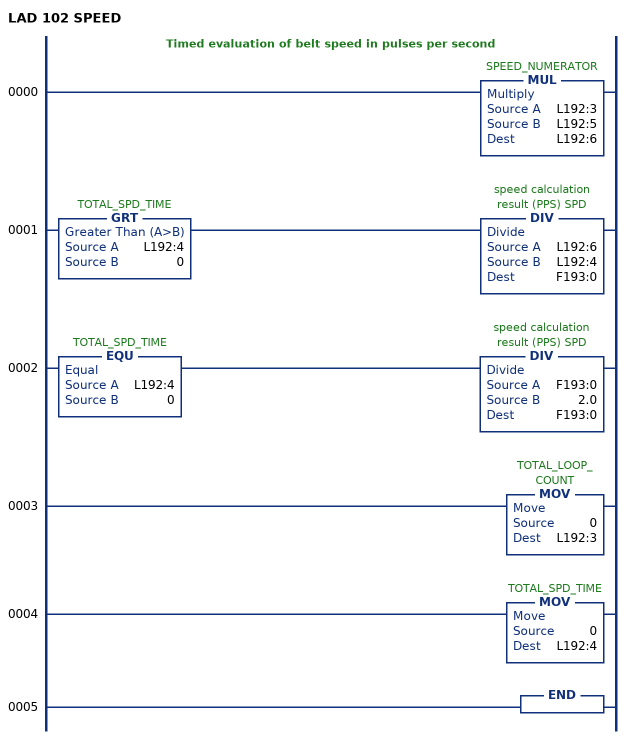
% Rung: 0 %
% TITLE: Timed evaluation of belt speed in pulses per second %
SOR MUL L192:3 L192:5 L192:6 EOR
%   L192:3  TOTAL_LOOP_COUNT %
%   L192:5  TKS_PER_SECOND %
%   L192:6  SPEED_NUMERATOR %
% Rung: 1 %
SOR GRT L192:4 0 DIV L192:6 L192:4 F193:0 EOR
%   L192:4  TOTAL_SPD_TIME %
%   L192:6  SPEED_NUMERATOR %
%   F193:0  SPD  "speed calculation result (PPS)" %
% Rung: 2 %
SOR EQU L192:4 0 DIV F193:0 2.0 F193:0 EOR
%   L192:4  TOTAL_SPD_TIME %
%   F193:0  SPD  "speed calculation result (PPS)" %
% Rung: 3 %
SOR MOV 0 L192:3 EOR
%   L192:3  TOTAL_LOOP_COUNT %
% Rung: 4 %
SOR MOV 0 L192:4 EOR
%   L192:4  TOTAL_SPD_TIME %
% Rung: 5 %
SOR END EOR

LADDER 104 "P ADJUST"
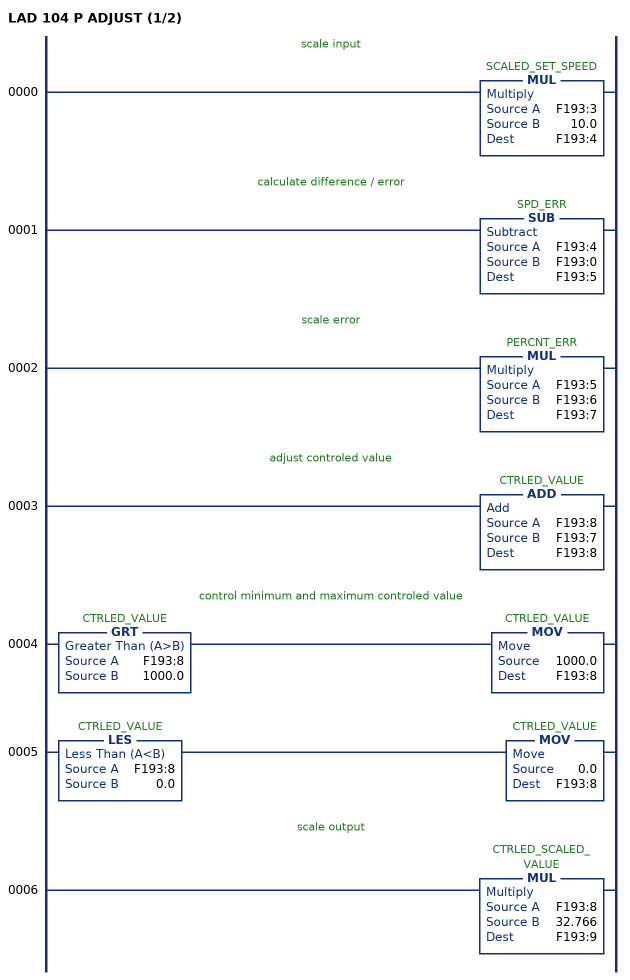
% Rung: 0 %
% scale input %
SOR MUL F193:3 10.0 F193:4 EOR
%   F193:3  SET_SPEED %
%   F193:4  SCALED_SET_SPEED %
% Rung: 1 %
% calculate difference / error %
SOR SUB F193:4 F193:0 F193:5 EOR
%   F193:4  SCALED_SET_SPEED %
%   F193:0  SPD  "speed calculation result (PPS)" %
%   F193:5  SPD_ERR %
% Rung: 2 %
% scale error %
SOR MUL F193:5 F193:6 F193:7 EOR
%   F193:5  SPD_ERR %
%   F193:6  FDBK_RATIO %
%   F193:7  PERCNT_ERR %
% Rung: 3 %
% adjust controled value %
SOR ADD F193:8 F193:7 F193:8 EOR
%   F193:8  CTRLED_VALUE %
%   F193:7  PERCNT_ERR %
% Rung: 4 %
% control minimum and maximum controled value %
SOR GRT F193:8 1000.0 MOV 1000.0 F193:8 EOR
%   F193:8  CTRLED_VALUE %
% Rung: 5 %
SOR LES F193:8 0.0 MOV 0.0 F193:8 EOR
%   F193:8  CTRLED_VALUE %
% Rung: 6 %
% scale output %
SOR MUL F193:8 32.766 F193:9 EOR
%   F193:8  CTRLED_VALUE %
%   F193:9  CTRLED_SCALED_VALUE %

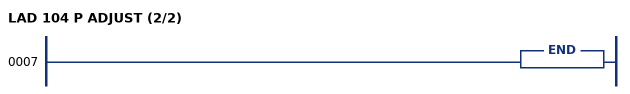
% Rung: 7 %
SOR END EOR

LADDER 110 "SHIFT"
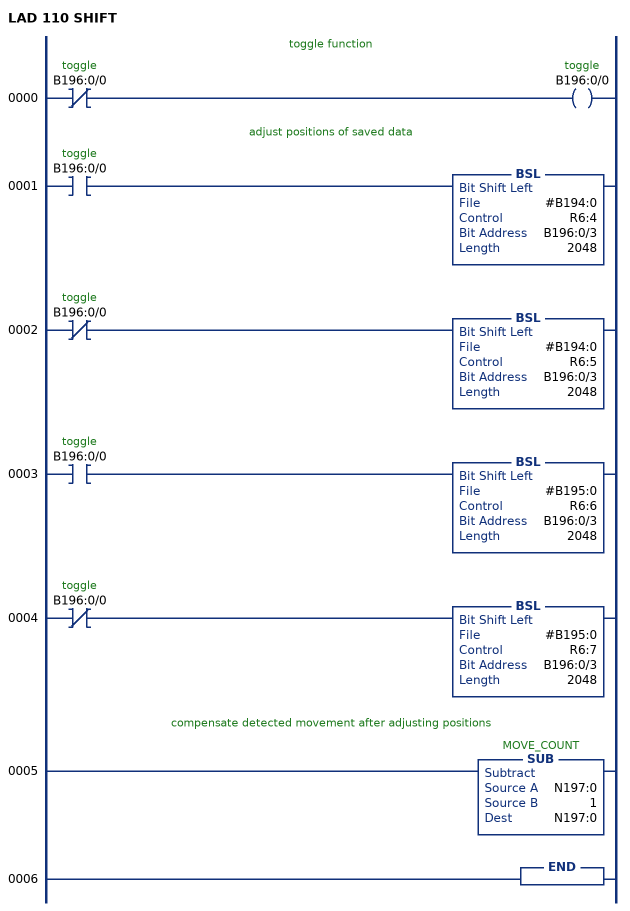
% Rung: 0 %
% toggle function %
SOR XIO B196:0/0 OTE B196:0/0 EOR
%   B196:0/0  "toggle" %
% Rung: 1 %
% adjust positions of saved data %
SOR XIC B196:0/0 BSL #B194:0 R6:4 B196:0/3 2048 EOR
%   B196:0/0  "toggle" %
%   B196:0/3  OFF %
% Rung: 2 %
SOR XIO B196:0/0 BSL #B194:0 R6:5 B196:0/3 2048 EOR
%   B196:0/0  "toggle" %
%   B196:0/3  OFF %
% Rung: 3 %
SOR XIC B196:0/0 BSL #B195:0 R6:6 B196:0/3 2048 EOR
%   B196:0/0  "toggle" %
%   B196:0/3  OFF %
% Rung: 4 %
SOR XIO B196:0/0 BSL #B195:0 R6:7 B196:0/3 2048 EOR
%   B196:0/0  "toggle" %
%   B196:0/3  OFF %
% Rung: 5 %
% compensate detected movement after adjusting positions %
SOR SUB N197:0 1 N197:0 EOR
%   N197:0  MOVE_COUNT %
% Rung: 6 %
SOR END EOR

LADDER 120 "SIM PARTS"
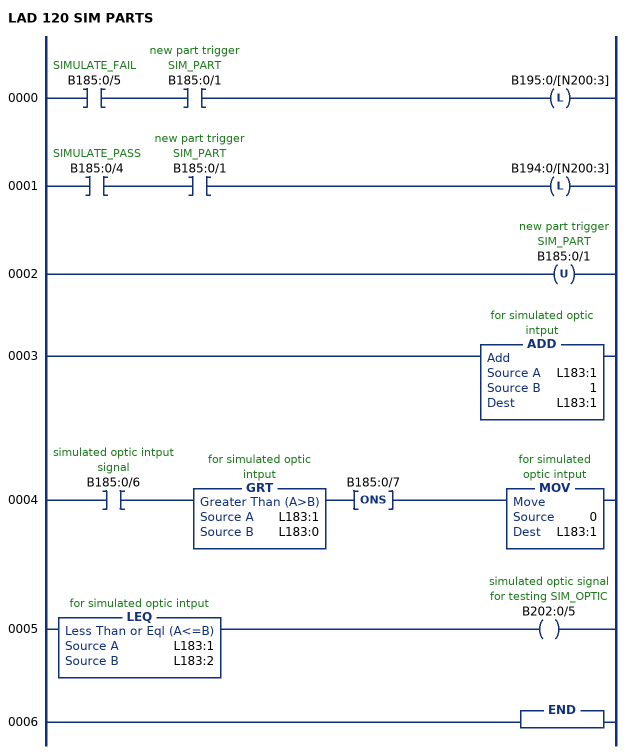
% Rung: 0 %
SOR XIC B185:0/5 XIC B185:0/1 OTL B195:0/[N200:3] EOR
%   B185:0/5  SIMULATE_FAIL %
%   B185:0/1  SIM_PART  "new part trigger" %
%   N200:3  OPT_LD_PT %
% Rung: 1 %
SOR XIC B185:0/4 XIC B185:0/1 OTL B194:0/[N200:3] EOR
%   B185:0/4  SIMULATE_PASS %
%   B185:0/1  SIM_PART  "new part trigger" %
%   N200:3  OPT_LD_PT %
% Rung: 2 %
SOR OTU B185:0/1 EOR
%   B185:0/1  SIM_PART  "new part trigger" %
% Rung: 3 %
SOR ADD L183:1 1 L183:1 EOR
%   L183:1  "for simulated optic intput" %
% Rung: 4 %
SOR XIC B185:0/6 GRT L183:1 L183:0 ONS B185:0/7 MOV 0 L183:1 EOR
%   B185:0/6  "simulated optic intput signal" %
%   L183:1  "for simulated optic intput" %
%   L183:0  "count for part data injection" %
% Rung: 5 %
SOR LEQ L183:1 L183:2 OTE B202:0/5 EOR
%   L183:1  "for simulated optic intput" %
%   L183:2  "simulated part width" %
%   B202:0/5  SIM_OPTIC  "simulated optic signal for testing" %
% Rung: 6 %
SOR END EOR

LADDER 121 "PARTDETECT"
